Staubli VAL3: page_editTraj.pjx

--- page_editTraj.pjx ---
Parameters version=s7.8.3 stackSize=10000 millimeterUnit=true
Program file=buildList.pgx
Program file=changePoint.pgx
Program file=goTo.pgx
Program file=insertInstr.pgx
Program file=listAdd.pgx
Program file=loadEditTraj.pgx
Program file=loadPage.pgx
Program file=main.pgx
Program file=onBackEvent.pgx
Program file=onEnterEvent.pgx
Program file=onExit.pgx
Program file=onF1Event.pgx
Program file=onF2Event.pgx
Program file=onF3Event.pgx
Program file=onF4Event.pgx
Program file=onF5Event.pgx
Program file=onF6Event.pgx
Program file=onF7Event.pgx
Program file=onF8Event.pgx
Program file=onSpaceEvent.pgx
Program file=onStart.pgx
Program file=password.pgx
Program file=refresh.pgx
Program file=refreshDynamic.pgx
Program file=refreshStatic.pgx
Program file=saveIt.pgx
Program file=selectItem.pgx
Program file=setAllAccel.pgx
Program file=setAllBlend.pgx
Program file=setAllSpeed.pgx
Program file=showPoint.pgx
Program file=showStatus.pgx
Program file=unSelectItem.pgx
Data file=page_editTraj.dtx
Library alias=use path=Disk://public_temp/userPage/userPage.pjx
Library alias=pub path=Disk://public_temp/pub/pub.pjx
Library alias=data path=Disk://SaveData/SaveData.pjx
Library alias=cycle path=Disk://cycle/cycle.pjx

--- page_editTraj.dtx ---
bool bButton[8]
  [0] = true
  [1] = true
  [2] = true
  [4] = true
  [5] = true
  [6] = true
  [7] = true
bool bExit
bool bLarge
bool bShowStatus
bool bTrigger
num nClockStatus = 962.397
num nIndex
num nIndexItem
num nKey
num nOldIndex
public num nPage
num nRefresh = 1149.353
num nSelected = -1
num nTime = 0.1
num nUserItem = 6
num nView
string sAction[3]
string sEvent = "Name: > appro"
public string sItems = "pick"
string sListUser[6]
  [0] = "appro   X > 0   "
  [1] = "appro   Y > 0   "
  [2] = "appro   Z > -50   "
  [3] = "appro  RX > 0   "
  [4] = "appro  RY > 0   "
  [5] = "appro  RZ > 0   "
string sMenu[8]
  [0] = "Here"
  [1] = "Align"
  [2] = "Tool"
  [4] = "Motion"
  [5] = "Delete"
  [6] = "Insert"
  [7] = "Save"
string sMenu8[8]
string sMenuUser[8]
  [0] = "Here"
  [1] = "Align"
  [2] = "Tool"
string sMessage[2]
  [0] = "ON"
  [1] = "OFF"
string sOldListUser
string sTrajName = "pick"
frame fFather = {fatherId=world[0]}
string sWorkingmode[16]
  [0] = "点属性      >"
  [1] = "Appro X     >"
  [2] = "Appro Y     >"
  [3] = "Appro Z     >"
  [4] = "Appro RX    >"
  [5] = "Appro RY    >"
  [6] = "Appro RZ    >"
  [7] = "速度        >"
  [8] = "加速度      >"
  [9] = "偏移方式    >"
  [10] = "偏移对象    >"
  [11] = "移动方式    >"
  [12] = "停止        >"
  [13] = "混合        >"
  [14] = "信号        >"
  [15] = "提前输出    >"
string sList
num i
public string sTitle
public string sPassword[2]
  [0] = "chenpeng"
  [1] = "xixi"
string sPasswd

--- main.pgx ---
public program main()
  local bool l_bSave
  local bool l_bOverRide
  local num l_nSize
  local bool l_bUnreached
  local string l_sMessage
  local bool l_bExit
  local string l_sEmpty
begin
  // INIT
  call onStart()
  // LOOP UNTIL Exit
  l_bExit=false
  do

    call refresh()
    nKey=getKey()
    call use:listevent(nKey,nIndex,sEvent)
    nView=use:nView
    nSelected=nIndex

    switch nKey
      case 270
        call onEnterEvent()
      break
      case 271
        call onF1Event()
      break
      case 272
        call onF2Event()
      break
      case 273
        call onF3Event()
      break
      case 274
        call onF4Event()
      break
      case 275
        call onF5Event()
      break
      case 276
        call onF6Event()
      break
      case 277
        call onF7Event()
      break
      case 278
        call onF8Event()
      break
      case 255
        l_bExit=true
      break

    endSwitch
    // release the resource
    delay(0)
    if workingMode()!=1
      call use:timerDialog("请切换成手动模式",0)
      wait(workingMode()==1)
    endIf
  until nKey==255
  use:bUseRefresh=true
  // on Exit
 // call onExit()
end

--- buildList.pgx ---
program buildList()
  local num l_nSize
  local num i
  local string l_sInstruction
  local string l_sMessage
  local string l_sTemp
  local string l_sEmpty
  local string l_sData
  local string l_sType
begin
  call use:setSizeList(13,0,25,9)
  //建立对话款
  call use:listcreate("")
//  l_sEmpty=""
  call use:stringCopy(l_sEmpty,sList)
//  call use:selectNewField(nSelected,nIndex,nView)
  call listAdd("点属性 "+">取片点移动")
  call listAdd("Appro "+" X  > "+toString(".2",data:pPoinTest[data:nPage_Traj].trsf.x))
  call listAdd("Appro "+" Y  > "+toString(".2",data:pPoinTest[data:nPage_Traj].trsf.y))
  call listAdd("Appro "+" Z  > "+toString(".2",data:pPoinTest[data:nPage_Traj].trsf.z))
  call listAdd("Appro "+" RX > "+toString(".2",data:pPoinTest[data:nPage_Traj].trsf.rx))
  call listAdd("Appro "+" RY > "+toString(".2",data:pPoinTest[data:nPage_Traj].trsf.ry))
  call listAdd("Appro "+" RZ > "+toString(".2",data:pPoinTest[data:nPage_Traj].trsf.rz))
  call listAdd("速度 "+" > "+toString(".2",data:mNomSpeed.vel)+"%")
  call listAdd("加速度 "+" > "+toString(".2",data:mNomSpeed.accel)+"%")
  call listAdd("偏移方式  >Appro")
  call listAdd("偏移对象  >摆正点")
  call listAdd("移动方式  >直线")
  call listAdd("停止  >[ ]")
  call listAdd("混合  >[ ]")
  call listAdd("输出提前 > 0mm")
  call use:listadd(sList)
 // nIndex=data:nPage_viewTraj
  call use:selectNewField(nSelected,nIndex,nView)
  call use:listupdate(0)
end

--- changePoint.pgx ---
program changePoint(num x_nIndex)
  local num i
  local string l_sMessage[3]
  local num l_nLocal
  local bool l_bOk
  local num l_nStop
  local string l_sButton[2]
  local string l_sEmpty
  local string l_sItem
  local string l_sData
  local string l_sPath
begin

end

--- goTo.pgx ---
program goTo(num x_nIndex, bool& x_bUnreached[])
  local bool l_bUnreached
  local num l_nIndexTool
  local tool l_tTool
begin
end

--- insertInstr.pgx ---
program insertInstr()
  local num i
  local string l_sMessage
  local num l_nIndex
  local string l_sItem
  local string l_sPath
begin
end

--- listAdd.pgx ---
program listAdd(string x_sEvent)
begin
    // add in the queue
  if sList!=""
    $dins(sList,size(sList))
  endIf
  sList[size(sList)-1]=x_sEvent
end

--- loadEditTraj.pgx ---
program loadEditTraj(string x_sName)
  local num i
  local num l_nIndex
  local string l_sPath
begin
end

--- loadPage.pgx ---
program loadPage(string x_sPage, string& x_sItems[])
// load the next page
  local num i
  local string l_sMessage
begin
end

--- onBackEvent.pgx ---
program onBackEvent(bool& x_bSave[])
  local num i
  local string l_sMessage[3]
  local num l_nLocal
  local bool l_bYes
  local string l_sAction[3]
  local num l_nIndex
  local string l_sButton[2]
begin

end

--- onEnterEvent.pgx ---
program onEnterEvent()
  local string l_sEmpty
  local string l_s
begin
  call use:findPos(sEvent,">",i)
  i=i+1
  if i!=-1
    l_sEmpty=""
    call use:listcursor(use:nView,false)
    switch nIndex
      case 0
        popUpMsg(sEvent)
      break
      case 1
        call use:changeValue(data:pPoinTest[data:nPage_Traj].trsf.x,-400,400,i+40-use:nBottomX,use:nView+1,l_sEmpty)
      break
      case 2
        call use:changeValue(data:pPoinTest[data:nPage_Traj].trsf.y,-400,400,i+40-use:nBottomX,use:nView+1,l_sEmpty)
      break
      case 3
        call use:changeValue(data:pPoinTest[data:nPage_Traj].trsf.z,-400,400,i+40-use:nBottomX,use:nView+1,l_sEmpty)
      break
      case 4
        call use:changeValue(data:pPoinTest[data:nPage_Traj].trsf.rx,-100,100,i+40-use:nBottomX,use:nView+1,l_sEmpty)
      break
      case 5
        call use:changeValue(data:pPoinTest[data:nPage_Traj].trsf.ry,-100,100,i+40-use:nBottomX,use:nView+1,l_sEmpty)
      break
      case 6
        call use:changeValue(data:pPoinTest[data:nPage_Traj].trsf.rz,-100,100,i+40-use:nBottomX,use:nView+1,l_sEmpty)
      break
    endSwitch
  endIf
    // set data
  call buildList()
  // save it
  data:libSave()



end

--- onExit.pgx ---
program onExit(bool& x_bSave[])
  local string l_sMessage
  local bool l_bYes
  local bool l_bCancel
  local string l_sButton[2]
begin

end

--- onF1Event.pgx ---
program onF1Event()
begin
  // look if the bButton is enable
  if bButton[0]
    //
    call password()
  endIf
end

--- onF3Event.pgx ---
program onF3Event()
begin
  // look if the bButton is enable
  if bButton[2]
    //
  endIf
end

--- onF4Event.pgx ---
program onF4Event()
  local string l_sMessage
  local num l_nActual
  local num l_nOldValue
  local num l_nX
  local num l_nY
begin
  // look if the bButton is enable
  if bButton[3]
    //
    //
    //
  endIf
end

--- onF5Event.pgx ---
program onF5Event()
  local string l_sMessage
  local num l_nActual
  local num l_nOldValue
  local num l_nMoveType
  local num l_nIndex
  local num l_nKey
  local string l_sEvent
begin
end

--- onF6Event.pgx ---
program onF6Event()
  local string l_sMessage
  local bool l_bYes
  local num l_nSize
  local num l_nFound
  local string l_sEvent
  local string l_sButton[2]
  local num l_nItem
begin
end

--- onF7Event.pgx ---
program onF7Event()
  local num l_nItem
begin

end

--- onF8Event.pgx ---
program onF8Event()
  local num i
  local num l_nResult
 begin
  // look if the bButton is enable
  if bButton[7]
    //
    call use:timerDialog("数据正在保存中....",1)
    call cycle:save(l_nResult)
    if l_nResult==0
      call use:timerDialog("数据已经保存成功",1)
    elseIf l_nResult!=0
      call use:timerDialog("数据未保存成功",1)
    endIf
  endIf
end

--- onSpaceEvent.pgx ---
program onSpaceEvent(bool& x_bSave[])
  local num i
  local string l_sMessage[3]
  local num l_nLocal
  local bool l_bYes
  local string l_sAction[3]
  local num l_nIndex
  local bool l_bStop
begin
end

--- onStart.pgx ---
program onStart()
  local num i
  local num l_nIndex
  local bool l_bOk
begin
  cls()
  // reset the Key pressure
  call use:nullKey(nKey)
  setTextMode(0)
  // build the list
  call buildList()
  nRefresh=clock()
 call refreshStatic()
end

--- password.pgx ---
program password()
begin
  cls()
  call use:timerDialog("请输入密码",0)
  call use:type(2,8,">>>>>")
  call use:read(3,8,sPasswd,15,true)

  if sPasswd==sPassword[0]
    sTitle=":true"
    popUpMsg("密码已经被修改")
  else
    sTitle=":false"
    popUpMsg("密码错误不能修改")
  endIf
  call buildList()
end

--- refresh.pgx ---
program refresh()
// // page refresh
begin
  if (nKey>=270 and nKey<=278) or use:bUseRefresh
    cls()
    call refreshStatic()
    call buildList()
    call refreshDynamic()
  else
    //refresh the Dynamic message
    if (clock()-nRefresh>nTime)
      call refreshDynamic()
    endIf
  endIf
  delay(0.1)
end

--- refreshDynamic.pgx ---
program refreshDynamic()
begin
    // DO NOT CHANGE
  nRefresh=clock()
  use:bUseRefresh=false
  //
  // ADD HERE
  //
end

--- refreshStatic.pgx ---
program refreshStatic()
  local string l_sMenu
  local num i
  local string l_sInstruction
  local num l_nSize
  local string l_sMessage
  local mdesc l_mDesc
  local num l_nTcpAction
  local string l_sName
  local string l_sEmpty
  local bool l_bStop
  local num l_nEmpty
  local num l_nIndexTool
  local string l_sType
  local string l_sData
begin
 // cls()
  title("编辑-1号石墨舟A面取片-第1槽/6槽")
  l_sMenu="权限,,,,,吸片,放片,保存"
  // define the menu
  call use:stringToArray(l_sMenu,sMenu)
  sMenu[0]=sMenu+sTitle
  call use:setMenu(sMenu,true,2)

////  call use:listadd(sList)



//  //
//  l_sMenu="1,2,,,,,,"
//  call use:stringToArray(l_sMenu,sMenu)
//  call use:setMenu(sMenu,false,3)
//  call use:getMenu(sMenu,bButton)

//  call use:setSizeList(0,0,38,12)
//  call use:listcreate("第1槽/8槽")
//  //
//  call use:listadd(sList)
//  //
//  // refresh the list
//  call use:selectNewField(nSelected,nIndex,nView)
//  //

//    title("111")
//    l_sMenu="模拟,复位,,,,,,"
//  // define the menu
//  call use:stringToArray(l_sMenu,sMenu)
//    // set the menu
//  call use:setMenu(sMenu,true,2)
//  call use:getMenu(sMenu,bButton)
end

--- saveIt.pgx ---
program saveIt(bool& x_bSave[])
  local string l_sMessage
  local num l_nResult
  local string l_sResult
begin
end

--- selectItem.pgx ---
public program selectItem(num x_nIndex)
  local string l_sItem
begin
end

--- setAllAccel.pgx ---
public program setAllAccel(num x_nNewValue, num x_nOldValue)
  local num i
  local num l_nSize
begin
end

--- setAllBlend.pgx ---
public program setAllBlend(num x_nNewValue, num x_nOldValue)
  local num i
  local num l_nSize
begin
end

--- setAllSpeed.pgx ---
program setAllSpeed(num x_nNewValue, num x_nOldValue)
  local num i
  local num l_nSize
begin
end

--- showPoint.pgx ---
program showPoint()
  local point l_pPoint[2]
  local num l_nIndexTool
  local tool l_tTool
  local point l_pHere
  local num i
  local joint l_jHere
begin
end

--- showStatus.pgx ---
program showStatus()
  local joint l_jHere
  local point l_pHere
  local string l_sMessage[2]
  local tool l_tTool
  local num l_nIndexTool
begin
end

--- unSelectItem.pgx ---
program unSelectItem()
  local string l_sEvent
  local num i
  local num l_nSize
begin
end
